FUNCTION_BLOCK AOI_WoodBunkAlarms
VAR_OUTPUT
	panelPowerOn : BOOL;
	safetyOk : BOOL;
	airPressureOk : BOOL;
END_VAR
VAR_OUTPUT
	alarm : BOOL;
END_VAR

alarm :=
	NOT panelPowerOn OR 
	NOT safetyOk OR
	NOT airPressureOk;

END_FUNCTION_BLOCK

(* stored: Version 1.1.0.1, ProductVersion 3.1.4024.11
   POU AOI_WoodBunkAlarms: Id {52cc73a4-5d87-414b-9f82-1691c8b1fc45}, SpecialFunc None *)
